FUNCTION_BLOCK SifbTimer
  (* Standard: 61499-2 *)
  (* Version 0.1, 2019-00-29, hpea485, UOA *)
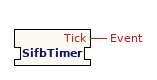
  EVENT_OUTPUT
    Tick;
  END_EVENT
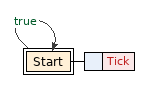
  EC_STATES
    Start : -> Tick;
  END_STATES
  EC_TRANSITIONS
    Start TO Start := true;
  END_TRANSITIONS
END_FUNCTION_BLOCK
